FUNCTION_BLOCK Rosca_HMI (* Service Interface Function Block Type *)
  (* Standard: 61499-2 *)
  (* Version 0.0, 04/03/2026, template *)
  PACKAGE Hidryco.HidrycoLib;
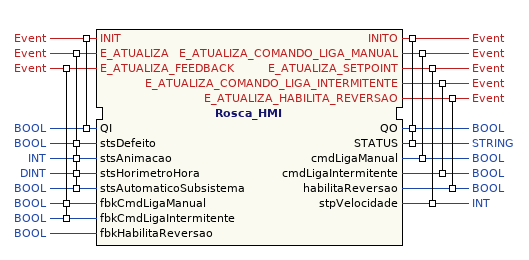
  EVENT_INPUT
    INIT WITH QI;
    E_ATUALIZA WITH stsDefeito, stsAnimacao, stsHorimetroHora, stsAutomaticoSubsistema;
    E_ATUALIZA_FEEDBACK WITH fbkCmdLigaManual, fbkCmdLigaIntermitente;
  END_EVENT
  EVENT_OUTPUT
    INITO WITH QO, STATUS;
    E_ATUALIZA_COMANDO_LIGA_MANUAL WITH cmdLigaManual;
    E_ATUALIZA_SETPOINT WITH stpVelocidade;
    E_ATUALIZA_COMANDO_LIGA_INTERMITENTE WITH cmdLigaIntermitente;
    E_ATUALIZA_HABILITA_REVERSAO WITH habilitaReversao;
  END_EVENT
  VAR_INPUT
    QI : BOOL;
    stsDefeito : BOOL;
    stsAnimacao : INT;
    stsHorimetroHora : DINT;
    stsAutomaticoSubsistema : BOOL;
    fbkCmdLigaManual : BOOL;
    fbkCmdLigaIntermitente : BOOL;
    fbkHabilitaReversao : BOOL;
  END_VAR
  VAR_OUTPUT
    QO : BOOL; (* Event Output Qualifier *)
    STATUS : STRING; (* Service Status *)
    cmdLigaManual : BOOL;
    cmdLigaIntermitente : BOOL;
    habilitaReversao : BOOL;
    stpVelocidade : INT;
  END_VAR
  SERVICE /
    SEQUENCE 
    END_SEQUENCE
  END_SERVICE
END_FUNCTION_BLOCK
